// TIA Portal V20 export
// export: Created 2026-10-03T18:54:34.1966347Z, ExportSetting WithDefaults, DisplayName Totally Integrated Automation Portal, DisplayVersion V20 Update 4, DisplayName TIA Portal Openness, DisplayVersion V20 Update 4, DisplayName TIA Portal Version Control Interface, DisplayVersion V20 Update 4, DisplayName SINAMICS Startdrive Advanced, DisplayVersion V20 SP1 Update 1, DisplayName SINAMICS Startdrive G110M, G120, G120C, G120D, G120P, G115D, DisplayVersion V20 SP1 Update 1, DisplayName SINAMICS Startdrive G130, G150, S120, S150, SINAMICS MV, G220, S200, S210, DisplayVersion V20 SP1 Update 1, DisplayName STEP 7 Professional, DisplayVersion V20 Update 4, DisplayName STEP 7 Safety, DisplayVersion V20 Update 2, DisplayName WinCC Basic/Comfort/Advanced, DisplayVersion V20 Update 4, DisplayName WinCC Unified, DisplayVersion V20 Update 4
FUNCTION "SLC_COP_MIXED" : Void   // FC11, SCL
TITLE = SLC COP between a float file and a B/N file
{ S7_Optimized_Access := 'TRUE' }
VERSION : 0.1
// Replaces a COP between a floating point file and a bit/integer file, which copies the raw words without
//  converting the values (typically to pass floats through integer registers to a SCADA or other system).
//  Length counts destination elements, as in the SLC. Note that TIA stores the high word of a float first;
//  check that the receiver expects that word order.
// stored: AutoNumber true, IsIECCheckEnabled false, SetENOAutomatically false, UDAEnableTagReadback false
   VAR_INPUT
      SrcFile : DInt;   // Source data file number
      SrcElement : DInt;   // First source element
      SrcIsFloat : Bool;   // TRUE if the source is an F file (4 bytes per element)
      DstFile : DInt;   // Destination data file number
      DstElement : DInt;   // First destination element
      DstIsFloat : Bool;   // TRUE if the destination is an F file (4 bytes per element)
      Length : DInt;   // Number of destination elements
   END_VAR
   VAR_TEMP
      srcSize : DInt;
      dstSize : DInt;
   END_VAR
BEGIN
   // Element sizes: 4 bytes for a float, 2 for a bit/integer word.
   IF #SrcIsFloat THEN #srcSize := 4; ELSE #srcSize := 2; END_IF;
   IF #DstIsFloat THEN #dstSize := 4; ELSE #dstSize := 2; END_IF;

   // 16#84 is the DB memory area.
   POKE_BLK(area_src := 16#84, dbNumber_src := #SrcFile, byteOffset_src := #SrcElement * #srcSize,
            area_dest := 16#84, dbNumber_dest := #DstFile, byteOffset_dest := #DstElement * #dstSize,
            count := #Length * #dstSize);
END_FUNCTION
